// TwinCAT 3 PLC project Untitled1
// ProgramVersion: 3.1.4023.0
// libraries:
//   stdNOV, * (National Oilwell Varco)
//   Tc2_FTP, * (Beckhoff Automation GmbH)
//   Tc2_Standard, * (Beckhoff Automation GmbH)
//   Tc2_System, * (Beckhoff Automation GmbH)
//   Tc2_Utilities, * (Beckhoff Automation GmbH)
//   Tc3_JsonXml, * (Beckhoff Automation GmbH)
//   Tc3_Module, * (Beckhoff Automation GmbH)
// project tree:
//   DUTs/ ST_ReceivedData.TcDUT
//   / PlcTask.TcTTO
//   POUs/ForceLimiter/ ForceLimiterControls.TcPOU, ForceLimiterFsmAction.TcDUT, ForceLimiterFSM.TcPOU, ForceLimiterFsmEvent.TcDUT, ForceLimiterFsmState.TcDUT
//   POUs/JsonParsing/ FTP_to_Beckhoff.TcPOU, ParseJsonDoc.TcPOU
//   POUs/LinearInterpolating/ LinearInterpolation.TcPOU
//   POUs/ MAIN.TcPOU

CONFIGURATION Untitled1
    RESOURCE PLC ON TwinCAT3
        TASK PlcTask(INTERVAL := T#10ms, PRIORITY := 20);
        PROGRAM MAIN WITH PlcTask : MAIN;
    END_RESOURCE
END_CONFIGURATION

// ---- DUTs/ST_ReceivedData.TcDUT
TYPE ST_ReceivedData :
STRUCT
	serialNumber 	: STRING(255);
	batteryVoltage 	: STRING(255);
	clickType		: STRING(255);
	ProjectInfo 	: STRING(255);
	ProjectName 	: STRING(255);
	UTCUnixDateTime : STRING(255);
	UpperPercent	: LREAL;
	LowerPercent	: LREAL;
// Unit Array
	uDepth : STRING(255);
	uRIH_SurfaceWt_CatastrophicBuckling : STRING(255);
	uRIH_SurfaceWt_FrictionPlus : STRING(255);
	uRIH_SurfaceWt : STRING(255);
	uRIH_SurfaceWt_FrictionNgtv : STRING(255);
	uPOOH_SurfaceWt_FrictionNgtv : STRING(255);
	uPOOH_SurfaceWt : STRING(255);
	uPOOH_SurfaceWt_FrictionPlus : STRING(255);
	uPOOH_SurfaceWt_Yield : STRING(255);
	
//Friction Data Array
	
	Depth			: ARRAY [1..50] OF LREAL;
	RIH_SurfaceWt_CatastrophicBuckling : ARRAY [1..50] OF LREAL;
	RIH_SurfaceWt_FrictionPlus : ARRAY [1..50] OF LREAL;
	RIH_SurfaceWt : ARRAY [1..50] OF LREAL;
	RIH_SurfaceWt_FrictionNgtv : ARRAY [1..50] OF LREAL;
	POOH_SurfaceWt_FrictionNgtv : ARRAY [1..50] OF LREAL;
	POOH_SurfaceWt : ARRAY [1..50] OF LREAL;
	POOH_SurfaceWt_FrictionPlus : ARRAY [1..50] OF LREAL;
	POOH_SurfaceWt_Yield	: ARRAY [1..50] OF LREAL;
END_STRUCT
END_TYPE

// ---- POUs/ForceLimiter/ForceLimiterFsmAction.TcDUT
TYPE ForceLimiterFsmAction :
(
	FsmAction_None := stdNOV.FSM_ACTION_NONE,	
	FsmAction_Warn,
	FsmAction_Crit_Alarm,	
	FsmAction_Clear_Warning,
	FsmAction_Clear_Crit_Alarm,	
	NUM_FsmActions
) BYTE;
END_TYPE

// ---- POUs/ForceLimiter/ForceLimiterFsmEvent.TcDUT
TYPE ForceLimiterFsmEvent :
(
	FsmEvent_Manual_Limits_Not_Set := 0,
	FsmEvent_Manual_Limits_Set,
	FsmEvent_Approaching_Limits,
	FsmEvent_Not_Approaching_Limits,
	FsmEvent_Limit_Surpassed,	
	FsmEvent_Limit_Not_Surpassed,	
	NUM_FsmEvents	
) BYTE;
END_TYPE

// ---- POUs/ForceLimiter/ForceLimiterFsmState.TcDUT
TYPE ForceLimiterFsmState :
(
	FsmState_Error := 0,
	FsmState_Off,
	FsmState_On,
	NUM_FsmStates
)BYTE;
END_TYPE

// ---- POUs/MAIN.TcPOU
(***********************************************************************
	Project:  Smart Injector
	Copyright (c) 2021 NOV AACD
	9720 Beechnut St
	Houston, TX  77036
	Phone: 936-777-6200
	Programmer: Mark Chandler <MDC>
	
	--------------------------------------------------------------------
	This software is the confidential and proprietary information of
	NOV AACD.("Confidential Information").  You shall not disclose such
	Confidential Information and shall use it only in accordance with
	the terms of the license agreement you entered into with NOV AACD.
	--------------------------------------------------------------------
	
	Code Name: 	MAIN
	Purpose:	Main PRG for Smart Injector
	
	Input values: NONE
	Output Values: NONE
	Revision: 0.1
	
	NOTES

	Jun 16 2021 - JW
	Added 'LinearInterpolation' FB for Cerberus data linear interpolation
	Added public properties to 'ParseJsonDoc' FB For accessing the Cererus data
	
	Mar 29 2021 - MDC
	MAIN complete for now
	Alarms System patched up with a fix in the library
	Testing of basic "Drivers" almost complete - need AO and encoder
	Prepped older code for deletion by removing from compilation, will delete after drivers finished
	I/O setup for testing only
	
	Mar 2 2021 - MDC
	Basic Methods, Structs, GVLs set up to support compilation for MAIN
	Security code omitted for now
	Most code ported from Wago
	Alarms need work
	 

	Feb 8 2021 - MDC
	Starting point for Smart Injector based on Ideal Frac Code and NOV Wiki
	https://wiki.nov.com/pages/viewpage.action?spaceKey=AACD&title=AACDRD-888+-+Cruise+Control+Project+Requirements
	Most basic code remains from Ideal Frac. Any Modbus or NSA references have been removed.

****************************************************************************)

PROGRAM MAIN
VAR
//////////////FTP Test Function Call//////////////////////////////////////////
	FTP_Test : FTP_to_Beckhoff;
	ParseJsonDoc1 : ParseJsonDoc ;

/////////////Linear Interpolation Call/////////////////////////////////////////
	receivedData						: ST_ReceivedData;
	Depth								: ARRAY [1..50] OF LREAL;
	RIH_SurfaceWt_CatastrophicBuckling 	: ARRAY [1..50] OF LREAL;
	RIH_SurfaceWt_FrictionPlus 			: ARRAY [1..50] OF LREAL;
	RIH_SurfaceWt 						: ARRAY [1..50] OF LREAL;
	RIH_SurfaceWt_FrictionNgtv 			: ARRAY [1..50] OF LREAL;
	POOH_SurfaceWt_FrictionNgtv 		: ARRAY [1..50] OF LREAL;
	POOH_SurfaceWt 						: ARRAY [1..50] OF LREAL;
	POOH_SurfaceWt_FrictionPlus 		: ARRAY [1..50] OF LREAL;
	POOH_SurfaceWt_Yield				: ARRAY [1..50] OF LREAL;

	StartFTP		: BOOL;
	LoadJsonData	: BOOL;
	JsonDataLoaded  : BOOL;
	CerberusData1	: LinearInterpolation;	
	CerberusData2	: LinearInterpolation;
	actualDepth		: LREAL;	// Actual depth value
	RIH_SurfaceWtLP : LREAL;	// Calculated rih surface weight 
	POOH_SurfaceWtLP: LREAL;	// Calculated pooh surface weight
	RIH_CriticalWtLP: LREAL; 	// Calculated rih critical weight
	POOH_CriticalWtLP: LREAL;	// Calculated pooh surface weight
	
	
	Calculated		: BOOL;		// Output is calculated
	Error			: BOOL;		// X-values sequence is wrong
	BelowLower 		: BOOL;		// Input value is below lower range
	OverUpper  		: BOOL;		// Input value is over upper range
	
	// Force Limiter Controls
	forceLimiter1		: ForceLimiterControls;
	// INPUT
	rih					: BOOL;		// Run in hole
	pooh				: BOOL;		// Pull out of hole
	cruiseControl		: BOOL; 	// Cruise control mode
	autoMill			: BOOL;		// Auto mill mode
	cerberusDataLoaded 	: BOOL;		// Cerberus data loaded
	surfaceWeight		: LREAL;	// Actual surface weight (lbs)	
	maxSnub				: LREAL; 	// Max Sbub (in negative lbs)
	maxPull				: LREAL;	// Max Pull (lbs)
	criticalWeightRih	: LREAL;	// RIH critical weight (Cerburus Catastrophic Buckling, in negative lbs)
	criticalWeightPooh	: LREAL;	// POOH critical weight ( Cerburus 80% pipe yield force, lbs)
	exitAutoPercent		: LREAL:= 5.0;		// If surface weight exceed the Max Snub/Pull value by %, then exit automation mode
	exitAutoTiming		: TIME := T#10S;	// If surface weight exceed the Max Snub/Pull value over an interval, then exit automation mode		
	// OUTPUT
	surfaceWeightLow	: BOOL;		// Warning if surface weight is below the Max Snub
	surfaceWeightHigh	: BOOL;		// Warning if surface weight is over the Max Pull	
	reduceForce			: BOOL;		// Fast stop while POOH, or run at slow speed while RIH
	exitAuto			: BOOL;		// Exit automation if surface weight exceed the Max Snub/Pull values by percentage or over an interval	
END_VAR

// Develop Security Code AT a later DATE  - Mar 2 2021 <MDC>	
// Commissioning Code Generation	
(*	CommissionTrigger(CLK:= xCommission OR gstProcessData.PlcCommissionTrigger);
	IF (CommissionTrigger.Q) THEN
		WriteCommissionCode();
	END_IF *)
	
// Function Block Call
FTP_Test.Start := StartFTP;
FTP_Test(); 

// Function Block Call 
ParseJsonDoc1.loadJsonData := LoadJsonData;
ParseJsonDoc1();
LoadJsonData := ParseJsonDoc1.loadJsonData;

// Implement Linear Interpolation for Cerberus Data
JsonDataLoaded						:= ParseJsonDoc1.JsonDataLoaded;
receivedData 						:= ParseJsonDoc1.CerberusData;
Depth 								:= receivedData.Depth;
RIH_SurfaceWt_CatastrophicBuckling 	:= receivedData.RIH_SurfaceWt_CatastrophicBuckling;
RIH_SurfaceWt_FrictionPlus			:= receivedData.RIH_SurfaceWt_FrictionPlus;
RIH_SurfaceWt						:= receivedData.RIH_SurfaceWt;
RIH_SurfaceWt_FrictionNgtv			:= receivedData.RIH_SurfaceWt_FrictionNgtv;
POOH_SurfaceWt_FrictionNgtv			:= receivedData.POOH_SurfaceWt_FrictionNgtv;
POOH_SurfaceWt						:= receivedData.POOH_SurfaceWt;
POOH_SurfaceWt_FrictionPlus			:= receivedData.POOH_SurfaceWt_FrictionPlus;
POOH_SurfaceWt_Yield				:= receivedData.POOH_SurfaceWt_Yield;

IF ParseJsonDoc1.numOfPoints >= 2 AND ParseJsonDoc1.numOfPoints <= 50 THEN
	CerberusData1(lrX := actualDepth, 
				 arrX := Depth, 
		   	    arrY1 := RIH_SurfaceWt, 
		        arrY2 := POOH_SurfaceWt, 
	     usiNumOfElem := ParseJsonDoc1.numOfPoints, 
			     lrY1 => RIH_SurfaceWtLP, 
			     lrY2 => POOH_SurfaceWtLP, 
		        bCalc => Calculated, 
			     bErr => Error, 
	      bLowerLimit => BelowLower, 
	      bUpperLimit => OverUpper);
	
	CerberusData2(lrX := actualDepth, 
				 arrX := Depth, 
		   	    arrY1 := RIH_SurfaceWt_CatastrophicBuckling, 
		        arrY2 := POOH_SurfaceWt_Yield, 
	     usiNumOfElem := ParseJsonDoc1.numOfPoints, 
			     lrY1 => RIH_CriticalWtLP, 
			     lrY2 => POOH_CriticalWtLP);	  
		  
END_IF

// Implement Force Limiter Controls
forceLimiter1(Rih  				:= rih,
			  Pooh 				:=pooh,
			  CruiseControl 	:= cruiseControl,
			  AutoMill 			:= autoMill,
			  CerberusDataLoaded:= JsonDataLoaded,
			  SurfaceWeight		:= surfaceWeight,
			  MaxSnub			:= maxSnub,
			  MaxPull   		:= maxPull,
			  CriticalWeightRih := RIH_CriticalWtLP,
			  CriticalWeightPooh:= POOH_CriticalWtLP,
			  ExitAutoPercent 	:= 5.0,
			  ExitAutoTiming 	:= T#10S,
			  SurfaceWeightLow 	=> surfaceWeightLow,
			  SurfaceWeightHigh => surfaceWeightHigh,
			  ReduceForce 		=> reduceForce,
			  ExitAuto 			=> exitAuto);

END_PROGRAM

// ---- POUs/JsonParsing/FTP_to_Beckhoff.TcPOU
FUNCTION_BLOCK FTP_to_Beckhoff
(*create a user with the username "TestUser" AND the password"Test123" on the FTP Server. 
If you set a rising edge at the variable "startstop", the downloading will be
started. 

Notice that the user "TestUser" has rights FOR reading AND writing.*)
VAR
	RisingEdge : R_TRIG;
	startstop : BOOL;
	state : BYTE;
	FB_FTP_Open1 : FB_FTP_Open;
	FB_FTP_FileDownload1 : FB_FTP_FileDownload;
	FB_FTP_Close1 : FB_FTP_Close;
	JsonParsInsit : FB_JsonDynDomParser;
	//List_Param1 : ST_FTP_ConnInfo;
	JSON_FileOpen : FB_FileOpen;
	JSON_FileRead : FB_FileRead;
	list : ARRAY [0..5] OF ST_FTP_ConnInfo;
	FB_FTP_Info1 : FB_FTP_Info;
	busy : BOOL;
	err : BOOL;
	errid : UDINT;
	handle : T_HFTP;
	progress : UDINT;
	Samples: INT;
	TF6300: INT;
	cbList : UDINT;
	Counter: UINT;
	JSONArrayMember: FB_JsonDomParser;
	TriggerJSONCall : BOOL := TRUE;
END_VAR

VAR_INPUT
	//sNetID: T_AmsNetID;	
END_VAR

(***********************************************************************
	Project:  [Template]
	Copyright (c) 2016 NOV CTES
	3770 Pollok Dr
	Conroe, TX  77303
	Phone: 936-777-6200
	Programmer: Richard Koontz
	
	--------------------------------------------------------------------
	This software is the confidential and proprietary information of
	NOV CTES.("Confidential Information").  You shall not disclose such
	Confidential Information and shall use it only in accordance with
	the terms of the license agreement you entered into with NOV CTES.
	--------------------------------------------------------------------
	
	Code Name: 	FTP Connection Info and Data Transfer 

	Purpose:	
	
	Input values: NONE
	Return Value: NONE
	Revision: NONE
*************************************************************************)

// - At first a connection to a FTP Server will be opened with the function block FB_FTP_Open. 
RisingEdge(CLK:= startstop);
IF RisingEdge.Q THEN
	state := 1;
END_IF

CASE state OF
0:
	;
// Getting connection information with the FB_FTP_Info
//Error Information
	// - errid =33318: Requested action not taken. File unavailable (e.g., file not found, no access)
	// - errid =6: Target port not found – ADS server is not started or is not reachable
1:
FB_FTP_Info1(
	sNetID	:= '192.168.4.81.1.1', 				// sNetID is a string containing the AMS network identifier of the target device to which the ADS command is directed
	pList:= ADR(list),       					// Pointer address to a variable of the type ST_FTP_ConnInfo. This variable can also be an array of the type ST_FTPConnInfo
	cbList := SIZEOF(list),
	bExecute:= TRUE, //startstop,						// The command is executed with the rising edge
	tTimeout := T#15S,  						// States the time before the function is cancelled.
	bBusy=> busy, 								// The command is in the process of being transmitted by ADS. No new command will be accepted as long as "bBusy" remains TRUE.
	bError => err,								// Becomes TRUE, as soon as an error occurs.
	nErrID => errid);							// Supplies the ErrorCode
IF NOT busy AND NOT err THEN						 	//AND NOT err THEN
	FB_FTP_Info1(bExecute:= FALSE);
	State := 2;
END_IF  


// - At first a connection to a FTP Server will be opened with the function block FB_FTP_Open. 
2:
FB_FTP_Open1(
	sNetID:= '192.168.4.81.1.1',   			// sNetID is a string containing the AMS network identifier of the target device to which the ADS command is directed
	sHost:= '192.168.4.200',					//172.16.9.223 Is a string containing the IPv4 address of the FTP-Server
	nPort:= 21,									// FTP port (default 21)
	sUsername:= 'CAN-5CD9037LN9\TestUser', 		// CAN-5CD90910x6\ Username for the FTP Server authentication
	sPassword:= 'Test123', 						// Password for the FTP Server authentication
	bExecute:= TRUE,							// The command is executed with the rising edge.
	tTimeout:= T#15S,							// States the time before the function is cancelled.
	bBusy=> busy,
	bError=> err,
	nErrId=> errid,
	hFTP=> handle);
IF NOT busy AND NOT err THEN
	FB_FTP_Open1(bExecute:= FALSE);
	state := 3;
END_IF

// - After that the given file "\TestFolder\File1.txt" from the FTP Server will be downloaded with the function block FB_FTP_FileDownload.
// - The following path "\Program Files\TestFile1.txt" is the place where the file will be stored on the ADS device.
3:
FB_FTP_FileDownload1(
	sNetID:= '192.168.4.81.1.1',				// Is a string containing the AMS network identifier of the target device to which the ADS command is directed.
	hFTP:= handle,								// Handle to a FTP Server
	sSrcFile:= 'JSON_Testing.json',	// Source file which will be copied from the FTP Server
	sDesFile:= 'C:\FTP Test\JSON_Testing.json', // Path and name of the destination file on the ADS device
	bExecute:= TRUE,
	tTimeout:= T#15S,
	bBusy => busy,
	bError => err,
	nErrId => errid,
	nProgress => progress);
IF NOT busy AND NOT err THEN							//AND NOT err THEN
	FB_FTP_FileDownload1(bExecute:= FALSE);
	state := 4;
END_IF

// - At the end the connection to the FTP Server will be closed with the function block FB_FTP_Close.
4:
FB_FTP_Close1(
	sNetID:= '192.168.4.81.1.1',			 	// Is a string containing the AMS network identifier of the target device to which the ADS command is directed.
	hFTP:= handle,								// Handle to a FTP Server
	bExecute:= TRUE,
	tTimeout:= T#15S,
	bBusy => busy,
	bError => err,
	nErrId => errid);
IF NOT busy AND NOT err THEN 				//AND NOT err THEN
	FB_FTP_Close1(bExecute:= FALSE);
	state := 0;
END_IF
END_CASE

PROPERTY PUBLIC Start : BOOL
SET
startstop := Start;
END_SET
END_PROPERTY

END_FUNCTION_BLOCK

// ---- POUs/JsonParsing/ParseJsonDoc.TcPOU
FUNCTION_BLOCK ParseJsonDoc
VAR
	(* JSON *)
	fbJson 			: FB_JsonDomParser();
	fbJsonSax		: FB_JsonSaxReader();
	jsonProp		: SJsonValue;
	jsonValue		: SJsonValue;
	bHasMember		: BOOL;
  	sMessage 		: STRING(255) := '{"serialNumber":"G030PT028191AC4R","batteryVoltage":"1547mV","clickType":"SINGLE"}';
	stReceivedData	: ST_ReceivedData;
	
	//sPath			: STRING := 'C:\FTP Test\JSON_Testing.json'; // PLC path
	sPath			: STRING := 'C:\Users\wuj2\OneDrive - NOV Inc\Documents\_Projects\Cerberus\JSON_Testing.json'; // Local path for testing
	bLoaded			: BOOL;
	bLoad			: BOOL;
	count			: INT;
	sDoc			: STRING(255);
	bDataLoaded		: BOOL;	// Data loaded flag
	
	bIsArray 		: BOOL;
	jsonIterator	: SJsonValue;
	jsonIteratorEnd	: SJsonValue;
	sName 			: SJsonValue;
	jsonArray 		: sJsonValue;
	CopyJsonDoc 	: UDINT;
	pJsonDoc 		: STRING(15000);
	nJsonDoc 		: UDINT;
	ReadJsonCount 	: INT;
	MaxArrayCount 	: INT := 43;
	JsonDateTime 	: BOOL;
	nFT 			: FILETIME;
	DecodeFileTime	: INT;
	jsonDoc			: SJsonValue; //ULINT;
	dateTime		: INT;
	nDT 			: DATE_AND_TIME;
	sDT				: STRING := '1611612069.019';
	
	i 				: USINT;
	NumOfMember		: USINT; // The number of points to interpolate
END_VAR

// Reset data loaded flag
IF bLoad = TRUE THEN
	bDataLoaded := FALSE;
END_IF

(* Retrieve JSON content *)
bLoaded := fbJson.LoadDocumentFromFile(sFile:=sPath , bExec:=bLoad);
//sDoc := fbJson.GetDocument();
CopyJsonDoc := fbJson.CopyDocument( pJsonDoc, SIZEOF(pJsonDoc));
IF bLoaded = TRUE THEN
	count 		:= count + 1	;
	bDataLoaded := TRUE;
END_IF

jsonDoc := fbJson.ParseDocument(pJsonDoc);
//CopyJsonDoc := fbJson.CopyDocument( pJsonDoc, SIZEOF(20000));

// reading simple JSON array
// Reading Project Info Array from JSON Document 
		bHasMember := fbJson.HasMember(jsonDoc, 'ProjectInfo');
IF (bHasMember) THEN
	  bHasMember := FALSE;
	  	jsonArray := fbJson.FindMember(jsonDoc, 'ProjectInfo');
	  	bIsArray := fbJson.IsArray(jsonArray);
	  	jsonIterator := fbJson.ArrayBegin(jsonArray);
	  	sName:= fbJson.GetArrayValue(jsonIterator);
	  
	  // this way does it by member iteration
	  	jsonProp := fbJson.MemberBegin(sName);
	  	jsonValue := fbJson.GetMemberValue(jsonProp);
	  	stReceivedData.ProjectName := fbJson.GetString(jsonValue);
	  
	  	jsonProp := fbJson.FindMember(sName, 'UTCUnixDateTime');
	  	//stReceivedData.UTCUnixDateTime := fbJson.GetString(jsonProp);
	  	JsonDateTime := fbJsonSax.DecodeDateTime(sDT);
	  	jsonProp := fbJson.FindMember(sName, 'UpperPercent');
	  	stReceivedData.UpperPercent := fbJson.GetDouble(jsonProp);
	  
	  	jsonProp := fbJson.FindMember(sName, 'LowerPercent');
	  	stReceivedData.LowerPercent := fbJson.GetDouble(jsonProp);
	  
	  // this way does it by looking for a specific member
	  //jsonProp := fbJson.FindMember(sName, 'UpperPercent');
//stReceivedData.UpperPercent := fbJson.GetDouble(jsonProp);
	  
	END_IF

// Reading Units from JSON Document 
		bHasMember := fbJson.HasMember(jsonDoc, 'Units');
IF (bHasMember) THEN
	  	bHasMember := FALSE;
	  	jsonArray := fbJson.FindMember(jsonDoc, 'Units');
	  	bIsArray := fbJson.IsArray(jsonArray);
	  	jsonIterator := fbJson.ArrayBegin(jsonArray);
	  	sName	   := fbJson.GetArrayValue(jsonIterator);
	  
	  // this way does it by member iteration
	  	jsonProp := fbJson.MemberBegin(sName);
	  	jsonValue := fbJson.GetMemberValue(jsonProp);
	  	stReceivedData.uDepth := fbJson.GetString(jsonValue);
	  
	  	jsonProp := fbJson.FindMember(sName, 'uDepth');
	  	stReceivedData.uDepth := fbJson.GetString(jsonProp);
	  
	  	jsonProp := fbJson.FindMember(sName, 'uRIH_SurfaceWt_CatastrophicBuckling');
	  	stReceivedData.uRIH_SurfaceWt_CatastrophicBuckling := fbJson.GetString(jsonProp);
	  
	  	jsonProp := fbJson.FindMember(sName, 'uRIH_SurfaceWt_FrictionPlus');
	  	stReceivedData.uRIH_SurfaceWt_FrictionPlus := fbJson.GetString(jsonProp);
	  
	  	jsonProp := fbJson.FindMember(sName, 'uRIH_SurfaceWt');
	  	stReceivedData.uRIH_SurfaceWt_FrictionPlus := fbJson.GetString(jsonProp);
	  
	  	jsonProp := fbJson.FindMember(sName, 'uRIH_SurfaceWt_FrictionNgtv');
	  	stReceivedData.uRIH_SurfaceWt_FrictionNgtv := fbJson.GetString(jsonProp);
	  
	  	jsonProp := fbJson.FindMember(sName, 'uRIH_SurfaceWt_FrictionNgtv');
	  	stReceivedData.uRIH_SurfaceWt_FrictionNgtv := fbJson.GetString(jsonProp);
	  
	  	jsonProp := fbJson.FindMember(sName, 'uRIH_SurfaceWt_FrictionNgtv');
	  	stReceivedData.uRIH_SurfaceWt_FrictionNgtv := fbJson.GetString(jsonProp);
	  
	  	jsonProp := fbJson.FindMember(sName, 'uPOOH_SurfaceWt_FrictionNgtv');
	  	stReceivedData.uPOOH_SurfaceWt_FrictionNgtv := fbJson.GetString(jsonProp);
	  
	   	jsonProp := fbJson.FindMember(sName, 'uPOOH_SurfaceWt');
	  	stReceivedData.uPOOH_SurfaceWt := fbJson.GetString(jsonProp);
	  
	   	jsonProp := fbJson.FindMember(sName, 'uPOOH_SurfaceWt_FrictionPlus');
	  	stReceivedData.uPOOH_SurfaceWt_FrictionPlus := fbJson.GetString(jsonProp);
	  
	   	jsonProp := fbJson.FindMember(sName, 'uPOOH_SurfaceWt_Yield');
	  	stReceivedData.uPOOH_SurfaceWt_Yield := fbJson.GetString(jsonProp);

END_IF



//FOR ReadJsonCount := 1 TO MaxArrayCount  BY 1 DO
bHasMember := fbJson.HasMember(jsonDoc, 'FrictionData');
	
IF (bHasMember) THEN
	  	bHasMember := FALSE;
	  	jsonArray := fbJson.FindMember(jsonDoc, 'FrictionData');
	  	jsonIterator := fbJson.ArrayBegin(jsonArray);
		jsonIteratorEnd := fbJson.ArrayEnd(jsonArray);
		i := 1;
	WHILE jsonIterator <> jsonIteratorEnd DO
		sName := fbJson.GetArrayValue(jsonIterator);

	  	bIsArray := fbJson.IsArray(jsonArray);
	  	sName	   := fbJson.GetArrayValue(jsonIterator);
	  
	  	jsonProp := fbJson.MemberBegin(sName);
	  	jsonValue := fbJson.GetMemberValue(jsonProp);
	  	stReceivedData.Depth[i] := fbJson.GetDouble(jsonValue);
	  
	  	jsonProp := fbJson.FindMember(sName, 'RIH_SurfaceWt_CatastrophicBuckling');
	  	stReceivedData.RIH_SurfaceWt_CatastrophicBuckling[i] := fbJson.GetDouble(jsonProp);  
	  
	  	jsonProp := fbJson.FindMember(sName, 'RIH_SurfaceWt_FrictionPlus');
	  	stReceivedData.RIH_SurfaceWt_FrictionPlus[i] := fbJson.GetDouble(jsonProp);

	  	jsonProp := fbJson.FindMember(sName, 'RIH_SurfaceWt');
	  	stReceivedData.RIH_SurfaceWt[i] := fbJson.GetDouble(jsonProp);
	  
	  	jsonProp := fbJson.FindMember(sName, 'RIH_SurfaceWt_FrictionNgtv');
	  	stReceivedData.RIH_SurfaceWt_FrictionNgtv[i] := fbJson.GetDouble(jsonProp);
	  
	  	jsonProp := fbJson.FindMember(sName, 'POOH_SurfaceWt_FrictionNgtv');
	  	stReceivedData.POOH_SurfaceWt_FrictionNgtv[i] := fbJson.GetDouble(jsonProp);
	  
	  	jsonProp := fbJson.FindMember(sName, 'POOH_SurfaceWt');
	  	stReceivedData.POOH_SurfaceWt[i] := fbJson.GetDouble(jsonProp);
	  
	  	jsonProp := fbJson.FindMember(sName, 'POOH_SurfaceWt_FrictionPlus');
	  	stReceivedData.POOH_SurfaceWt_FrictionPlus[i] := fbJson.GetDouble(jsonProp);
	  
	  	jsonProp := fbJson.FindMember(sName, 'POOH_SurfaceWt_Yield');
	  	stReceivedData.POOH_SurfaceWt_Yield[i] := fbJson.GetDouble(jsonProp);

	  	jsonIterator := fbJson.NextArray(jsonIterator);
		
		IF i < 50 THEN
			i := i + 1;
		END_IF		
		
	END_WHILE
	NumOfMember := i - 1;  
	
END_IF

PROPERTY PUBLIC CerberusData : ST_ReceivedData
GET
CerberusData := stReceivedData;
END_GET
END_PROPERTY

PROPERTY PUBLIC JsonDataLoaded : BOOL
GET
JsonDataLoaded := bDataLoaded;
END_GET
END_PROPERTY

PROPERTY PUBLIC loadJsonData : BOOL
GET
loadJsonData := bLoad;
END_GET
SET
bLoad := loadJsonData;
END_SET
END_PROPERTY

PROPERTY PUBLIC numOfPoints : USINT
GET
numOfPoints := NumOfMember;
END_GET
END_PROPERTY

END_FUNCTION_BLOCK

// ---- POUs/LinearInterpolating/LinearInterpolation.TcPOU
FUNCTION_BLOCK LinearInterpolation
(* 
The function block 'LinearInterpolation' represents two linear interpolations with
up to 50 inierpolation points and can be used to generate two characteristic
curves. 

The interpolation points are determined via field variables (arrX[1]/arrY1[1] to
arrX[n]/arrY1[n], and arrX[1]/arrY2[1] to arrX[n]/arrY2[n]).

The input values for lrX[n+1] must always be at least 0.0000001 greater than
values for lrX[n].

The parameter for the number of interpolation points, usiNumOfElem, must be in 
range 2..50.
*)

VAR_INPUT
	lrX			: LREAL;					// Input value of the characteristic curve
	arrX		: ARRAY[1..50] OF LREAL;	// Field with the X-values for the interpolation points
	arrY1		: ARRAY[1..50] OF LREAL;	// Field with the Y1-values for the interpolation points
	arrY2		: ARRAY[1..50] OF LREAL;	// Field with the Y2-values for the interpolation points
	usiNumOfElem: USINT(2..50);				// Number of interpolation points, internally limited to values between 2 and 50	
END_VAR
VAR_OUTPUT
	lrY1		: LREAL;	// Calculated output Y1 of the characteristic curve
	lrY2		: LREAL;	// Calculated output Y2 of the characteristic curve
	bCalc		: BOOL;		// Output is calculated
	bErr		: BOOL;		// X-values sequence is wrong
	bLowerLimit : BOOL;		// Input value is below lower range
	bUpperLimit : BOOL;		// Input value is over upper range
END_VAR
VAR
	i			: USINT;		
	t			: LREAL;
END_VAR
VAR CONSTANT
	INPUT_VALUE_MIN_DIFF	: LREAL := 0.0000001;	
END_VAR

// Check input array sequence error
FOR i := 1 TO usiNumOfElem - 1 DO
	IF (arrX[i + 1] - arrX[i]) <= INPUT_VALUE_MIN_DIFF THEN
		bErr := TRUE;
		EXIT;
	ELSE
		bErr := FALSE;
	END_IF
END_FOR

IF bErr = FALSE THEN
	// Get the points for interpolating 
	IF lrX < arrX[1] THEN
		// If X value is below first point, use first two points for interpolating 
		bLowerLimit	:= TRUE;
		bUpperLimit	:= FALSE;
		bCalc  		:= TRUE;		
		t 	 		:= (lrX - arrX[1])/(arrX[2] - arrX[1]);
		lrY1 		:= (1 - t) * arrY1[1] + t * arrY1[2];
		lrY2 		:= (1 - t) * arrY2[1] + t * arrY2[2];
	ELSIF lrX > arrX[usiNumOfElem] THEN
		// If X value is over last point, use last two points for interpolating
		bLowerLimit := FALSE;
		bUpperLimit := TRUE;
		bCalc  		:= TRUE;		
		t 	 		:= (lrX - arrX[usiNumOfElem - 1])/(arrX[usiNumOfElem] - arrX[usiNumOfElem - 1]);
		lrY1 		:= (1 - t) * arrY1[usiNumOfElem - 1] + t * arrY1[usiNumOfElem];
		lrY2 		:= (1 - t) * arrY2[usiNumOfElem - 1] + t * arrY2[usiNumOfElem];		
	ELSE
		bLowerLimit := FALSE;
		bUpperLimit := FALSE;
		FOR i := 1 TO usiNumOfElem - 1 DO
			IF lrX = arrX[i] THEN
				bCalc  	:= FALSE;
				lrY1 := arrY1[i];
				lrY2 := arrY2[i];
				EXIT;
			ELSIF lrX > arrX[i] AND lrX < arrX[i + 1] THEN
				bCalc  	:= TRUE;
				t 	 	:= (lrX - arrX[i])/(arrX[i + 1] - arrX[i]);
				lrY1 	:= (1 - t) * arrY1[i] + t * arrY1[i + 1];
				lrY2 	:= (1 - t) * arrY2[i] + t * arrY2[i + 1];
				EXIT;
			END_IF			
		END_FOR
		
		IF lrX = arrX[usiNumOfElem] THEN
			bCalc  	:= FALSE;
			lrY1 := arrY1[usiNumOfElem];
			lrY2 := arrY2[usiNumOfElem];
		END_IF
		
	END_IF	
	
END_IF

END_FUNCTION_BLOCK

// ---- POUs/ForceLimiter/ForceLimiterControls.TcPOU
// Set job limits in terms of max snub and max pull
FUNCTION_BLOCK PUBLIC ForceLimiterControls
VAR_INPUT
	Rih					: BOOL;		// Run in hole
	Pooh				: BOOL;		// Pull out of hole
	CruiseControl		: BOOL; 	// Cruise control mode
	AutoMill			: BOOL;		// Auto mill mode
	CerberusDataLoaded 	: BOOL;		// Cerberus data loaded
	SurfaceWeight		: LREAL;	// Actual surface weight (lbs)	
	MaxSnub				: LREAL; 	// Max Sbub (in negative lbs)
	MaxPull				: LREAL;	// Max Pull (lbs)
	CriticalWeightRih	: LREAL;	// RIH critical weight (Cerburus Catastrophic Buckling, in negative lbs)
	CriticalWeightPooh	: LREAL;	// POOH critical weight ( Cerburus 80% pipe yield force, lbs)
	ExitAutoPercent		: LREAL:= 5.0;		// If surface weight exceed the Max Snub/Pull value by %, then exit automation mode
	ExitAutoTiming		: TIME := T#10S;	// If surface weight exceed the Max Snub/Pull value over an interval, then exit automation mode		
END_VAR
VAR_OUTPUT
	SurfaceWeightLow	: BOOL;		// Warning if surface weight is below the Max Snub
	SurfaceWeightHigh	: BOOL;		// Warning if surface weight is over the Max Pull	
	ReduceForce			: BOOL;		// Fast stop while POOH, or run at slow speed while RIH
	ExitAuto			: BOOL;		// Exit automation if surface weight exceed the Max Snub/Pull values by percentage or over an interval
END_VAR
VAR
	t_SurfaceWtLowMaxSnub	: BOOL;	// Surface weight below Max Snub
	t_SurfaceWtLowCritRih	: BOOL;	// Surface weight below Critical Weight RIH
	t_SurfaceWtHighMaxPull	: BOOL;	// Surface weight over Max Pull
	t_SurfaceWtHighCritPooh	: BOOL; // Surface weight over Critical Weight POOH
	t_SurfaceWtLowMaxTimer	: TON;	// Surface weight below the Max Snub timer
	t_SurfaceWtHighMaxTimer	: TON;	// Surface weight over the Max pull timer
	t_SurfaceWtLowEnough	: BOOL;	// Surface weight exceed max snub by percentage or timing
	t_SurfaceWtHighEnough	: BOOL;	// Surface weight exceed max pull by percentage or timing
END_VAR

// Run in hole
IF Rih = TRUE THEN
	// Surface weight below Max Snub	
	t_SurfaceWtLowMaxSnub := SurfaceWeight < MaxSnub;
	t_SurfaceWtLowMaxTimer(IN := t_SurfaceWtLowMaxSnub, PT := ExitAutoTiming);
	
	// 	Surface weight below critical weight RIH
	t_SurfaceWtLowCritRih := CerberusDataLoaded AND SurfaceWeight < CriticalWeightRih;
	
	// Warn surceface weight too low
	SurfaceWeightLow := t_SurfaceWtLowMaxSnub OR t_SurfaceWtLowCritRih;
	
	// Automation disable tolerance surpassed
	t_SurfaceWtLowEnough := SurfaceWeight < (1 + ExitAutoPercent / 100.0) * MaxSnub OR t_SurfaceWtLowMaxTimer.Q OR (MaxSnub = 0.0);
	
ELSE
	SurfaceWeightLow := FALSE;
	t_SurfaceWtLowMaxTimer(IN := FALSE);
	t_SurfaceWtLowEnough := FALSE;
END_IF

// Pull out of hole
IF Pooh = TRUE THEN
	// Surface weight over Max pull
	t_SurfaceWtHighMaxPull := SurfaceWeight > MaxPull;	
	t_SurfaceWtHighMaxTimer(IN := t_SurfaceWtHighMaxPull, PT := ExitAutoTiming);
	
	// Surface weight over Critical weight POOH	
	t_SurfaceWtHighCritPooh := CerberusDataLoaded AND SurfaceWeight > CriticalWeightPooh;
	
	// Warn surceface weight too high
	SurfaceWeightHigh := t_SurfaceWtHighMaxPull OR t_SurfaceWtHighCritPooh;
	
	// Automation disable tolerance surpassed
	t_SurfaceWtHighEnough := SurfaceWeight > (1 + ExitAutoPercent / 100.0) * MaxPull OR t_SurfaceWtHighMaxTimer.Q OR (MaxPull = 0.0);
ELSE
	SurfaceWeightHigh := FALSE;
	t_SurfaceWtHighMaxTimer(IN := FALSE);
	t_SurfaceWtHighEnough := FALSE;
END_IF

// Reduce force command and Disable automation
IF CruiseControl = TRUE OR AutoMill = TRUE THEN
	ReduceForce := SurfaceWeightLow OR SurfaceWeightHigh;
	ExitAuto	:= t_SurfaceWtLowEnough OR t_SurfaceWtHighEnough;
ELSE
	ReduceForce := FALSE;
	ExitAuto	:= FALSE;
END_IF

END_FUNCTION_BLOCK

// ---- POUs/ForceLimiter/ForceLimiterFSM.TcPOU
FUNCTION_BLOCK ForceLimiterFSM IMPLEMENTS i_actionHandler
VAR_INPUT
	xEnable				: BOOL;				// Enable inputs and FSM operation
	MaxSnub				: LREAL; 			// Max Sbub (in negative lbs)
	MaxPull				: LREAL;			// Max Pull (lbs)
	Rih					: BOOL;				// Run in hole
	Pooh				: BOOL;				// Pull out of hole
	CriticalWeightRih	: LREAL;			// RIH critical weight (Cerburus Catastrophic Buckling, in negative lbs)
	CriticalWeightPooh	: LREAL;			// POOH critical weight ( Cerburus 80% pipe yield force, lbs)	
	SurpassTimeout 		: TIME  := T#10S;	// Limit surpass timeout value input
	SurpassThreshhold	: LREAL := 3.0;		// Limit surpass threshhod in %	
	CerberusDataLoaded 	: BOOL;				// Cerberus data loaded
	SurfaceWeight		: LREAL;			// Actual surface weight (lbs)	
END_VAR
VAR_OUTPUT
	Warn		: BOOL;		// Approaching limits warn
	CritAlarm	: BOOL;		// Limits surpassed alarm	
	ReduceForce	: BOOL;		// Fast stop while POOH, or run at slow speed while RIH
	AutoDisable	: BOOL;		// Disable automation if surface weight exceed surpass limits
END_VAR
VAR
	(* Calcution mode *)
	m_Pull			: BOOL; 	// Pull caluculation mode, weight is positive
	m_SurfaceWeight : LREAL;	// Normalized surface weight
	m_SurpassLimit	: LREAL;	// Surpassed limit
	m_Limit			: LREAL;	// Limit
	m_ApproachLimit : LREAL;	// Approaching limit
	

	(* Event Triggers *)	
	m_EnableTrigger			: R_TRIG;	// Enable event trigger
	m_SurpassTimeOutTrigger	: R_TRIG;	// Limit surpass timeout event trigger
	m_SurpassTimer			: TON;		// Limit surpass timer used to detect timeout error


	(* Finite State Machine *)
	m_ForceLimiterFsmTable	: ARRAY[0..FSM_STATE_ARRAY_MAX, 0..FSM_EVENT_ARRAY_MAX, 0..FSM_ACTIONS_ARRAY_MAX] OF BYTE := [
	(* FsmState_Error --------------------------------------------------------- *)
	(*  Next State							Action								*)
	
		(* FsmEvent_Manual_Limits_Not_Set *)
		FSM_EVENT_INVALID,					ForceLimiterFsmAction.FsmAction_None,
		
		(* FsmEvent_Manual_Limits_Set *)
		FSM_EVENT_INVALID,					ForceLimiterFsmAction.FsmAction_None,
		
		(* FsmEvent_Approaching_Limits *)
		FSM_EVENT_INVALID,					ForceLimiterFsmAction.FsmAction_None,
		
		(* FsmEvent_Not_Approaching_Limits *)
		FSM_EVENT_INVALID,					ForceLimiterFsmAction.FsmAction_None,
		
		(* FsmEvent_Limit_Surpassed *)
		FSM_EVENT_INVALID,					ForceLimiterFsmAction.FsmAction_None,
		
		(* FsmEvent_Limit_Not_Surpassed *)
		FSM_EVENT_INVALID,					ForceLimiterFsmAction.FsmAction_None,	

	(* FsmState_Off ----------------------------------------------------------- *)
	(*  Next State							Action								*)
	
		(* FsmEvent_Manual_Limits_Not_Set *)
		ForceLimiterFsmState.FsmState_Off,	ForceLimiterFsmAction.FsmAction_Crit_Alarm,
		
		(* FsmEvent_Manual_Limits_Set *)
		ForceLimiterFsmState.FsmState_On,	ForceLimiterFsmAction.FsmAction_None,
		
		(* FsmEvent_Approaching_Limits *)
		ForceLimiterFsmState.FsmState_Off,	ForceLimiterFsmAction.FsmAction_None,
		
		(* FsmEvent_Not_Approaching_Limits *)
		ForceLimiterFsmState.FsmState_Off,	ForceLimiterFsmAction.FsmAction_None,
		
		(* FsmEvent_Limit_Surpassed *)
		ForceLimiterFsmState.FsmState_Off,	ForceLimiterFsmAction.FsmAction_None,
		
		(* FsmEvent_Limit_Not_Surpassed *)
		ForceLimiterFsmState.FsmState_Off,	ForceLimiterFsmAction.FsmAction_None,

	(* FsmState_On ------------------------------------------------------------ *)
	(*  Next State							Action								*)
	
		(* FsmEvent_Manual_Limits_Not_Set *)
		ForceLimiterFsmState.FsmState_Off,	ForceLimiterFsmAction.FsmAction_None,
		
		(* FsmEvent_Manual_Limits_Set *)
		ForceLimiterFsmState.FsmState_On,	ForceLimiterFsmAction.FsmAction_None,
		
		(* FsmEvent_Approaching_Limits *)
		ForceLimiterFsmState.FsmState_On,	ForceLimiterFsmAction.FsmAction_Warn,
		
		(* FsmEvent_Not_Approaching_Limits *)
		ForceLimiterFsmState.FsmState_On,	ForceLimiterFsmAction.FsmAction_Clear_Warning,
		
		(* FsmEvent_Limit_Surpassed *)
		ForceLimiterFsmState.FsmState_On,	ForceLimiterFsmAction.FsmAction_Crit_Alarm,
		
		(* FsmEvent_Limit_Not_Surpassed *)
		ForceLimiterFsmState.FsmState_On,	ForceLimiterFsmAction.FsmAction_Clear_Crit_Alarm	
	];

	m_ForceLimiterFSM : fb_FSM(	fsmId			:= ADR(	m_ForcelimiterFSM ),
								stateTable		:= ADR( m_ForceLimiterFsmTable ),
								actionHandler	:= THIS^,
								numStates		:= ForcelimiterFsmState.NUM_FsmStates,
								numEvents		:= ForceLimiterFsmEvent.NUM_FsmEvents,
								initialState	:= ForcelimiterFsmState.FsmState_Off);
								
	m_FsmError			: BOOL;					// FSM error bit (TRUE - FSM Halted)
	m_FsmErrorNum		: TFsmError;			// FSM error ENUM number
	m_FsmCurrentState	: ForceLimiterFsmState;	// Current FSM state output
	m_FsmLastState		: ForceLimiterFsmState; // Previous state used for debugging FSM errors
	m_FsmLastEvent		: ForceLimiterFsmEvent; // Last triggered event output
	m_FsmLastAction		: ForceLimiterFsmAction;// Last run action output	
END_VAR
VAR CONSTANT
	FSM_NUM_EVENT_ACTIONS	: INT := 1;
	FSM_NUM_STATES			: INT := ForceLimiterFsmState.NUM_FsmStates;
	FSM_NUM_EVENTS			: INT := ForceLimiterFsmEvent.NUM_FsmEvents;
	FSM_STATE_ARRAY_MAX		: INT := FSM_NUM_STATES - 1;
	FSM_EVENT_ARRAY_MAX		: INT := FSM_NUM_EVENTS - 1;
	FSM_ACTIONS_ARRAY_MAX	: INT := FSM_NUM_EVENT_ACTIONS;
END_VAR

// (* FSM *)

m_ForceLimiterFSM( xEnable := xEnable, xError => m_FsmError, errorNum => m_FsmErrorNum);

m_FsmCurrentState := m_ForceLimiterFSM.FSM_GetCurrentState();

IF Pooh = TRUE AND Rih = FALSE THEN
	m_Pull := TRUE;
ELSIF Pooh = FALSE AND Rih = TRUE THEN
	m_Pull := FALSE;
END_IF

// Pull operation 
IF m_Pull = TRUE THEN
	m_SurfaceWeight := SurfaceWeight;	
	IF CerberusDataLoaded = TRUE THEN
		m_Limit	:= MIN(MaxPull, CriticalWeightPooh);		
	ELSE 
		m_Limit	:= MaxPull;		
	END_IF
	m_SurpassLimit 	:= m_Limit * ( 1 + SurpassThreshhold / 100.0);		
	m_ApproachLimit := m_Limit * ( 1 - SurpassThreshhold / 100.0);	

// Snub operation	
ELSE
	m_SurfaceWeight := -1.0* SurfaceWeight;
	IF CerberusDataLoaded = TRUE THEN
		m_Limit	:= -1.0 * MAX(MaxSnub, CriticalWeightPooh);		
	ELSE 
		m_Limit	:= -1.0 * MaxSnub;		
	END_IF
	m_SurpassLimit 	:= -1.0 * MAX(MaxSnub, CriticalWeightPooh) * ( 1 + SurpassThreshhold / 100.0);		
	m_ApproachLimit := -1.0 * MAX(MaxSnub, CriticalWeightPooh) * ( 1 - SurpassThreshhold / 100.0);	
	
END_IF

// Timing if the surface weight is larger than the limit
m_SurpassTimer(IN := (m_SurfaceWeight > m_Limit), PT := SurpassTimeout);


// (* EVENT TRIGGER *)

// Reset FSM to initialization state
m_EnableTrigger(CLK := xEnable);
IF (m_EnableTrigger.Q) THEN
	m_ForceLimiterFSM.FSM_Reset();
END_IF

// Manual limits not set
IF MaxSnub >= 0.0 OR MaxPull <= 0.0 THEN
	m_ForceLimiterFSM.FSM_ProcessEvent(ForceLimiterFsmEvent.FsmEvent_Manual_Limits_Not_Set);
END_IF

// Manual limits set
IF MaxSnub < 0.0 AND MaxPull > 0.0 THEN
	m_ForceLimiterFSM.FSM_ProcessEvent(ForceLimiterFsmEvent.FsmEvent_Manual_Limits_Set);
END_IF

// Approaching the limit
IF m_SurfaceWeight >= m_ApproachLimit THEN
	m_ForceLimiterFSM.FSM_ProcessEvent(ForceLimiterFsmEvent.FsmEvent_Approaching_Limits);
ELSE
	m_ForceLimiterFSM.FSM_ProcessEvent(ForceLimiterFsmEvent.FsmEvent_Not_Approaching_Limits);
END_IF

// Surpassed the limit
IF m_SurfaceWeight >= m_SurpassLimit OR m_SurpassTimer.Q THEN
	m_ForceLimiterFSM.FSM_ProcessEvent(ForceLimiterFsmEvent.FsmEvent_Limit_Surpassed);
ELSE
	m_ForceLimiterFSM.FSM_ProcessEvent(ForceLimiterFsmEvent.FsmEvent_Limit_Not_Surpassed);
END_IF

METHOD ExcuteAction : BOOL
VAR_INPUT
	p_FSM			: POINTER TO fb_FSM;	// Pointer to the instatiation of the FSM object
	currentAction	: TFsmAction;			// Current FSM action being processed
	currentEvent	: TFsmEventDesc;		// Current FSM event being processed
END_VAR
CASE CurrentAction OF
	
	ForceLimiterFsmAction.FsmAction_None:	
		// Return TRUE
		ExcuteAction := TRUE;
		
	ForceLimiterFsmAction.FsmAction_Warn:	
		// Generate warn, reduce speed
		Warn		:= TRUE;		
		ReduceForce	:= TRUE;		
		
		// Return TRUE
		ExcuteAction := TRUE;
	
	ForceLimiterFsmAction.FsmAction_Crit_Alarm:
		// Generate critical alarm, disable cruise control and auto mill
		CritAlarm	:= TRUE;		
		AutoDisable	:= TRUE;		

		// Return TRUE
		ExcuteAction := TRUE;		
	
	ForceLimiterFsmAction.FsmAction_Clear_Warning:
		// Clear warning, reduce speed
		Warn		:= FALSE;		
		ReduceForce	:= FALSE;	
		
	ForceLimiterFsmAction.FsmAction_Clear_Crit_Alarm:
		// Clear critical alarm, enable cruise control and auto mill
		CritAlarm	:= FALSE;		
		AutoDisable	:= FALSE;		

		// Return TRUE
		ExcuteAction := TRUE;		
	
	FSM_ACTION_UNEXPECTED_EVENT:
		// Do action unexpected event
		p_FSM^.FSM_ASSERT(FALSE, TFsmError.FSM_INVALID_ACTION);
		
		// Return FALSE
		ExcuteAction := FALSE;
		
	FSM_ACTION_ERROR_EVENT:
		// Do action error event
		m_EnableTrigger(CLK := FALSE);
		
		// Return FALSE
		ExcuteAction := FALSE;

ELSE
	// Error trap - Unknow action
	p_FSM^.FSM_ASSERT(FALSE, TFsmError.FSM_INVALID_ACTION);
	
	// Return FALSE
	ExcuteAction := FALSE;

END_CASE

m_FsmLastState	:= p_FSM^.FSM_GetPreviousState();
m_FsmLastEvent	:= currentEvent.event;
m_FsmLastAction	:= currentAction;
END_METHOD

END_FUNCTION_BLOCK
